FUNCTION_BLOCK STEST_END
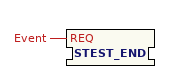
  EVENT_INPUT
    REQ;
  END_EVENT
END_FUNCTION_BLOCK
